// Identifies a Stage execution thread.
INTERFACE I_Thread EXTENDS _I_Thread

END_INTERFACE

(* stored: Version 1.1.0.1
   Itf I_Thread: Id {919f2c9a-a145-41ef-97f2-9f811fe90153} *)
